SUBAPPLICATION RequestOrchestrationOpcUaFull (* Request Orchestration using OPC UA with all fields from services, system and cloud to be set *)
  (* Standard: 61499-2; Description: Copyright (c) 2019 fortiss GmbH This program and the accompanying materials are made available under the terms of the Eclipse Public License 2.0 which is available at https://www.eclipse.org/legal/epl-2.0/ SPDX-License-Identifier: EPL-2.0 *)
  (* Version 1.0, 2019-09-17, Jose Cabral, fortiss GmbH *)
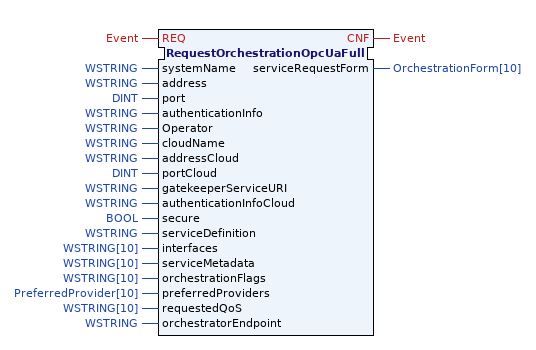
  EVENT_INPUT
    REQ; (* Request orchestration *)
  END_EVENT
  EVENT_OUTPUT
    CNF; (* Request finished *)
  END_EVENT
  VAR_INPUT
    systemName : WSTRING; (* Identification of the system *)
    address : WSTRING; (* Address of the offered services *)
    port : DINT; (* Port of the of the offered services *)
    authenticationInfo : WSTRING; (* Authentication info of the system *)
    Operator : WSTRING; (* Company (the capital  O is to avoid clash when exporting to C++) *)
    cloudName : WSTRING; (* Identification of the cloud *)
    addressCloud : WSTRING; (* Address to access the cloud *)
    portCloud : DINT; (* Port to access the cloud *)
    gatekeeperServiceURI : WSTRING; (* (Unclear documentation) *)
    authenticationInfoCloud : WSTRING; (* Authentication info of the cloud *)
    secure : BOOL; (* (Unclear documentation) *)
    serviceDefinition : WSTRING; (* Identification of the service *)
    interfaces : ARRAY [0..9] OF WSTRING; (* Interfaces implemented by the service *)
    serviceMetadata : ARRAY [0..9] OF WSTRING; (* Metadata of the service in key=value format *)
    orchestrationFlags : ARRAY [0..9] OF WSTRING; (* These flags can be set to tailor the orchestration process (use just the names of the flags to be enabled) *)
    preferredProviders : ARRAY [0..9] OF PreferredProvider; (* There can be a list from the Consumer stating which other Application Systems (even from other Clouds) it wishes to connect. If this field is filled out, the Orchestrator will try to facilitate these preferences *)
    requestedQoS : ARRAY [0..9] OF WSTRING; (* This object will be presenting the Consumer’s selected QoS level. Not implemented *)
    orchestratorEndpoint : WSTRING; (* Enpoint of the orchestrator *)
  END_VAR
  VAR_OUTPUT
    serviceRequestForm : ARRAY [0..9] OF OrchestrationForm; (* Response from the orchestrator *)
  END_VAR
  FBS
    FieldsToArrowheadCloud : FieldsToArrowheadCloud;
    FieldsToArrowheadSystem : FieldsToArrowheadSystem;
  END_FBS
  SUBAPPS
    RequestOrchestrationOpcUaPartial : RequestOrchestrationOpcUaPartial;
  END_SUBAPPS
  EVENT_CONNECTIONS
    REQ TO FieldsToArrowheadSystem.REQ;
    FieldsToArrowheadSystem.CNF TO FieldsToArrowheadCloud.REQ;
    FieldsToArrowheadCloud.CNF TO RequestOrchestrationOpcUaPartial.REQ;
    RequestOrchestrationOpcUaPartial.CNF TO CNF;
  END_CONNECTIONS
  DATA_CONNECTIONS
    systemName TO FieldsToArrowheadSystem.systemName;
    Operator TO FieldsToArrowheadCloud.Operator;
    address TO FieldsToArrowheadSystem.address;
    port TO FieldsToArrowheadSystem.port;
    authenticationInfo TO FieldsToArrowheadSystem.authenticationInfo;
    cloudName TO FieldsToArrowheadCloud.cloudName;
    addressCloud TO FieldsToArrowheadCloud.address;
    portCloud TO FieldsToArrowheadCloud.port;
    gatekeeperServiceURI TO FieldsToArrowheadCloud.gatekeeperServiceURI;
    authenticationInfoCloud TO FieldsToArrowheadCloud.authenticationInfo;
    secure TO FieldsToArrowheadCloud.secure;
    FieldsToArrowheadSystem.arrowheadSystem TO RequestOrchestrationOpcUaPartial.requesterSystem;
    FieldsToArrowheadCloud.arrowheadCloud TO RequestOrchestrationOpcUaPartial.requesterCloud;
    serviceDefinition TO RequestOrchestrationOpcUaPartial.serviceDefinition;
    interfaces TO RequestOrchestrationOpcUaPartial.interfaces;
    serviceMetadata TO RequestOrchestrationOpcUaPartial.serviceMetadata;
    orchestrationFlags TO RequestOrchestrationOpcUaPartial.orchestrationFlags;
    preferredProviders TO RequestOrchestrationOpcUaPartial.preferredProviders;
    requestedQoS TO RequestOrchestrationOpcUaPartial.requestedQoS;
    orchestratorEndpoint TO RequestOrchestrationOpcUaPartial.orchestratorEndpoint;
    RequestOrchestrationOpcUaPartial.serviceRequestForm TO serviceRequestForm;
  END_CONNECTIONS
END_SUBAPPLICATION
